Yaskawa INFORM job: KRIS1(-160_-90)07.JBI

/JOB
//NAME KRIS1(-160_-90)07
//POS
///NPOS 268,268,268,15,0,0
///TOOL 0
///POSTYPE PULSE
///PULSE
C00000=-1357,-104031,-113776,9484,62521,80538
C00001=-1357,-104031,-113776,9484,62521,80538
C00002=-36470,-76528,-106815,19279,71473,77234
C00003=-134470,-76528,-106815,19279,71473,77234
C00004=-174981,-50493,-90161,40064,84672,66854
C00005=-187879,-63712,-94262,49080,81916,61249
C00006=-186060,-71155,-91964,59790,82905,66762
C00007=-178869,-72848,-88692,57971,77164,66872
C00008=-178869,-73293,-87273,58169,76560,66435
C00009=-178869,-73560,-86246,58315,76140,66130
C00010=-178674,-73111,-86205,58218,76137,66246
C00011=-177360,-70267,-84836,57702,75706,66732
C00012=-178674,-73111,-86205,58218,76137,66246
C00013=-178674,-71838,-89995,57689,77779,67427
C00014=-187879,-63712,-94262,49080,81916,61249
C00015=-188382,-49930,-83952,49213,82654,61403
C00016=-188014,-50962,-81654,49243,81175,60803
C00017=-188014,-51673,-80691,49342,80537,60470
C00018=-188014,-51583,-80818,49329,80620,60513
C00019=-186548,-48975,-79328,48719,80176,60967
C00020=-188014,-51583,-80818,49329,80620,60513
C00021=-188014,-47372,-85350,48920,83933,62231
C00022=-182062,-62332,-92296,30199,64588,50507
C00023=-184090,-61700,-84500,30217,57788,46513
C00024=-184090,-62275,-83323,30540,56902,46238
C00025=-184090,-62207,-83473,30499,57013,46272
C00026=-182547,-59219,-81900,29317,56990,46927
C00027=-184090,-62207,-83473,30499,57013,46272
C00028=-182062,-62332,-92296,30199,64588,50507
C00029=-213458,-81436,-127572,45024,85737,46387
C00030=-213462,-137262,-127618,80891,60645,46377
C00031=-213462,-137262,-127618,80891,60645,46377
C00032=-213462,-137262,-127281,45256,60365,46369
C00033=-190178,-104312,-111371,30656,55898,55861
C00034=-182510,-123951,-113302,29184,45443,56133
C00035=-182510,-123446,-111392,29630,44641,55847
C00036=-182510,-123495,-111565,29589,44713,55873
C00037=-180510,-119420,-110276,27514,45182,57098
C00038=-182510,-123495,-111565,29589,44713,55873
C00039=-182510,-124409,-115363,28705,46354,56443
C00040=-219776,-105077,-106077,50090,64862,45838
C00041=-220601,-99189,-101769,50266,65553,45786
C00042=-220601,-99263,-100237,50600,64914,45410
C00043=-220601,-99258,-100424,50559,64990,45455
C00044=-218392,-97957,-99927,49618,64034,46123
C00045=-220601,-99258,-100424,50559,64990,45455
C00046=-219776,-105077,-106077,50090,64862,45838
C00047=-190178,-104312,-111371,30656,55898,55861
C00048=-229240,-109114,-135810,47014,82062,49329
C00049=-229240,-109114,-135810,47014,82062,49329
C00050=-195224,-66819,-119592,28790,78815,60275
C00051=-159578,-94739,-111578,14965,102577,71346
C00052=-157566,-87256,-71357,3912,80960,68626
C00053=-158237,-87274,-67249,3997,78461,68317
C00054=-158512,-86753,-64553,4040,77085,68177
C00055=-158512,-85902,-62577,4050,76306,68151
C00056=-159334,-88042,-63583,4126,75872,67853
C00057=-159947,-89575,-64280,4185,75546,67628
C00058=-158678,-86897,-63962,4060,76658,68106
C00059=-158401,-87046,-65688,4022,77628,68233
C00060=-157724,-87159,-69865,3934,80101,68545
C00061=-157573,-90681,-89077,3900,90084,68907
C00062=-157703,-92030,-92713,3898,91631,68910
C00063=-158377,-93978,-89476,3949,88678,68591
C00064=-158653,-94353,-86922,3974,86930,68442
C00065=-158653,-94065,-85585,3975,86257,68419
C00066=-158901,-94897,-86117,3998,86172,68332
C00067=-159738,-97484,-87119,4071,85502,68025
C00068=-158508,-94414,-86637,3961,86718,68485
C00069=-158233,-93872,-88035,3937,87841,68614
C00070=-157561,-92106,-91348,3883,90748,68930
C00071=-157550,-88189,-103730,3988,100358,69239
C00072=-157494,-88262,-105997,3987,101710,69297
C00073=-158163,-92718,-103752,3992,98079,68960
C00074=-158927,-96366,-102620,4029,95553,68625
C00075=-158927,-96520,-101690,4026,94903,68601
C00076=-158927,-96495,-101852,4026,95015,68605
C00077=-159979,-100458,-103367,4107,93966,68220
C00078=-158702,-95424,-101809,4010,95525,68699
C00079=-158425,-94019,-102865,4000,96880,68834
C00080=-157748,-89886,-105246,3989,100429,69172
C00081=-156260,-82084,-105550,20461,72444,69801
C00082=-137260,-84248,-120477,10166,77039,76482
C00083=-137260,-138866,-133764,10166,31487,76482
C00084=-31464,-162597,-133764,10166,12061,76482
C00085=11401,-148032,-125425,11667,35640,75771
C00086=126225,-114648,-117375,36487,17100,65054
C00087=160935,-140983,-109640,13468,75088,74332
C00088=169853,-118963,-84593,12681,69660,-86771
C00089=185015,-85467,-64977,10138,72568,-81037
C00090=186046,-86587,-63372,10054,70902,-80807
C00091=186046,-85672,-61299,10100,70108,-80875
C00092=186099,-85805,-61481,10085,70145,-80849
C00093=187639,-87511,-62050,9863,69435,-80354
C00094=183812,-88241,-67244,10331,72692,-81455
C00095=173907,-109296,-96285,11524,80966,-84205
C00096=165243,-81442,-84446,9619,88683,-83239
C00097=165243,-81286,-81084,9622,86723,-83389
C00098=165344,-81527,-80785,9608,86408,-83377
C00099=165344,-81401,-79599,9612,85752,-83428
C00100=165344,-81434,-79892,9611,85913,-83415
C00101=166373,-84175,-81092,9484,85132,-83124
C00102=163979,-82682,-81772,9785,86585,-83830
C00103=160654,-84295,-101618,10197,98198,-83833
C00104=158831,-94543,-102742,7696,93888,-81952
C00105=159073,-94488,-101668,7659,93239,-81911
C00106=159073,-94700,-100523,7653,92432,-81960
C00107=159073,-94669,-100714,7655,92565,-81952
C00108=160071,-98397,-102165,7522,91459,-81686
C00109=158831,-94357,-103427,7703,94400,-81921
C00110=161715,-86803,-103327,4886,98608,-77730
C00111=162141,-92472,-85533,-3463,86932,-68770
C00112=161818,-87798,-71417,-3733,80713,-68419
C00113=160875,-83714,-65601,-3665,79192,-68698
C00114=161375,-83882,-63363,-3725,77755,-68482
C00115=161375,-83186,-61665,-3733,77069,-68462
C00116=161375,-83302,-61946,-3731,77181,-68466
C00117=162606,-86103,-62964,-3849,76427,-68017
C00118=161375,-84160,-64056,-3722,78038,-68491
C00119=162005,-87841,-70029,-3758,79847,-68329
C00120=161949,-92223,-96357,-3744,93768,-68761
C00121=161804,-92637,-92737,-3704,91325,-68737
C00122=160782,-89227,-87327,-3611,89709,-69033
C00123=161425,-90912,-85851,-3665,87970,-68764
C00124=161425,-90690,-84578,-3665,87303,-68744
C00125=161425,-90728,-84781,-3665,87408,-68747
C00126=162412,-93603,-85938,-3751,86691,-68391
C00127=161425,-91016,-86520,-3665,88326,-68774
C00128=162058,-93372,-91608,-3722,90267,-68620
C00129=162002,-88104,-107646,-3859,102814,-69021
C00130=161873,-89540,-106233,-3806,101205,-69011
C00131=162580,-93883,-103932,-3818,97597,-68666
C00132=159915,-93477,-102438,-3577,96772,-69526
C00133=159915,-93839,-100899,-3567,95642,-69493
C00134=159915,-93799,-101099,-3568,95785,-69497
C00135=160794,-97042,-102371,-3639,94941,-69180
C00136=159915,-93165,-103472,-3585,97568,-69550
C00137=164885,-102201,-108421,-4002,96197,-67859
C00138=149595,-96211,-103761,-5489,101844,-74102
C00139=148895,-100989,-103442,-6283,96942,-74202
C00140=149006,-93113,-100988,-5479,101691,-74295
C00141=149599,-96300,-103483,-5484,101628,-74092
C00142=137295,-108190,-106060,-5698,94014,-77976
C00143=149608,-96287,-103789,-5489,101823,-74097
C00144=160720,-151449,-123129,-13814,72249,-68439
C00145=174899,-138237,-126795,1008,88740,-67536
C00146=163022,-96341,-102515,22398,105363,-76518
C00147=163017,-96713,-99258,22147,103326,-76913
C00148=166118,-105377,-102170,18852,96347,-77230
C00149=163022,-96736,-99152,22139,103253,-76925
C00150=162158,-93804,-96763,22109,103515,-77196
C00151=174925,-92085,-97088,18785,97864,-73864
C00152=167549,-101389,-103915,18999,98984,-76305
C00153=163194,-119427,-113025,19710,97619,-78016
C00154=163006,-95534,-87485,21597,97146,-78065
C00155=166449,-103981,-88986,17839,88165,-78380
C00156=167279,-118842,-91930,16839,77497,-71410
C00157=163006,-94576,-83573,21494,95359,-78388
C00158=162142,-91714,-81191,21448,95589,-78662
C00159=178049,-105864,-87645,15594,79224,-67328
C00160=171906,-113065,-93299,16245,80217,-69386
C00161=173072,-122981,-101575,-4997,88706,-65554
C00162=166636,-106884,-92426,-2568,94448,-67910
C00163=167630,-109607,-91139,-2502,92292,-67531
C00164=162194,-92631,-84353,657,102863,-69400
C00165=163060,-95514,-86735,782,102839,-69097
C00166=155875,-120106,-94474,-3152,88541,-71437
C00167=155875,-121766,-97691,-3153,89666,-71465
C00168=178442,-133591,-104623,-8068,82135,-63325
C00169=176542,-133362,-109369,-6755,86992,-64211
C00170=163036,-88875,-67291,2288,96831,-69180
C00171=159610,-85618,-62441,1680,95605,-70370
C00172=162086,-85813,-60042,2106,93969,-69554
C00173=162173,-84225,-60457,2128,95039,-69506
C00174=163038,-86971,-62872,2279,95091,-69211
C00175=151835,-92381,-62525,304,92274,-73022
C00176=151835,-95702,-69255,305,94709,-73016
C00177=163041,-94022,-81579,12660,98605,-75478
C00178=162985,-87715,-64806,21312,87868,-79725
C00179=162980,-85781,-60474,21324,86307,-80003
C00180=163244,-83528,-57038,21357,85347,-80079
C00181=162985,-85725,-60330,21325,86250,-80011
C00182=162122,-82990,-57905,21265,86391,-80297
C00183=171549,-75890,-53739,21771,84944,-77151
C00184=153122,-94015,-66237,20488,88162,-83220
C00185=168603,-127327,-105850,12339,78437,77405
C00186=149894,-144724,-110594,14594,75698,70467
C00187=126225,-114648,-117375,36487,17100,65054
C00188=118781,-153853,-134406,32592,23357,65054
C00189=12470,-167083,-125425,11667,16324,75771
C00190=-137258,-84249,-120477,10166,64820,76482
C00191=-160540,-100857,-113063,23155,68829,67581
C00192=-174981,-50493,-90161,40064,84672,66854
C00193=-187879,-63712,-94262,49080,81916,61249
C00194=-230671,-89591,-126680,64018,108053,56526
C00195=-230671,-150117,-126680,83924,107200,56526
C00196=-230671,-150117,-126680,83924,107200,56526
C00197=-230671,-150117,-126680,39809,88276,56526
C00198=-185677,-128245,-133585,38839,68006,71149
C00199=-143279,-154007,-127386,2438,36675,82296
C00200=-143590,-141394,-120265,2620,38778,82199
C00201=-143742,-142485,-120562,2786,38406,82105
C00202=-143590,-141570,-120589,2614,38886,82201
C00203=-202436,-119741,-113840,40114,62182,59763
C00204=-198557,-130318,-109753,40932,40025,50599
C00205=-196641,-131399,-103756,47310,28244,43457
C00206=-193242,-140218,-107458,47365,24899,43542
C00207=-143279,-154007,-127386,2438,36675,82296
C00208=-143372,-162538,-136969,2444,38193,82294
C00209=-143372,-162538,-136969,2444,38193,82294
C00210=-169193,-120980,-126540,32650,66176,77929
C00211=-162706,-113692,-115443,30259,61179,79142
C00212=-159565,-103232,-109234,28227,61475,80556
C00213=-143742,-142485,-120562,2786,38406,82105
C00214=-143590,-141570,-120589,2614,38886,82201
C00215=-133202,-124644,-116491,13354,48701,89198
C00216=-140045,-120904,-111840,33091,52219,88326
C00217=-147445,-115513,-104255,49921,56750,87686
C00218=-147948,-114087,-100063,56693,57074,88007
C00219=-151078,-112408,-101145,56872,59820,87990
C00220=-162706,-113692,-115443,30259,61179,79142
C00221=-169193,-120980,-126540,32650,66176,77929
C00222=-169193,-120980,-126540,32650,66176,77929
C00223=-169193,-120980,-126540,32650,66176,77929
C00224=-169193,-120980,-126540,32650,66176,77929
C00225=-189746,-144194,-133392,42604,68859,69788
C00226=-182215,-131283,-122466,40105,65254,71827
C00227=-178156,-121131,-115309,38344,64069,73249
C00228=-157379,-154126,-124637,33193,46204,76615
C00229=-155622,-153970,-121840,43876,49612,78686
C00230=-159534,-158630,-125101,47522,52653,77846
C00231=-179897,-166210,-133900,51769,64813,73191
C00232=-179897,-166210,-133900,51769,64813,73191
C00233=-179897,-166210,-133900,51769,64813,73191
C00234=-144017,-127352,-123370,33815,56946,88116
C00235=-136296,-120281,-120593,-4079,55650,85264
C00236=-135245,-107004,-113403,-4642,58094,85574
C00237=-145143,-100864,-111178,1649,59705,81829
C00238=-158741,-87238,-105999,9726,64424,77163
C00239=-147367,-98171,-102243,-17290,47874,78333
C00240=-144875,-102905,-108473,-14295,50590,79740
C00241=-136296,-120281,-120593,-4079,55650,85264
C00242=-138675,-113827,-131364,-2561,67962,83610
C00243=-184171,-107868,-119248,16468,98370,62097
C00244=-171634,-136713,-119987,14813,82155,64373
C00245=-158729,-95167,-103646,5818,103191,69841
C00246=-160167,-97375,-101626,5748,100928,69246
C00247=-158743,-95268,-103371,5812,102972,69826
C00248=-157888,-92366,-100981,5813,102933,70115
C00249=-149921,-107326,-105235,5663,97333,72568
C00250=-153886,-106740,-107354,5718,99208,71304
C00251=-163031,-143044,-118600,5591,88166,67691
C00252=-166711,-113552,-95038,4166,94777,66107
C00253=-164943,-103868,-87794,1353,97515,66988
C00254=-158755,-94787,-86481,-976,103949,69303
C00255=-157900,-91912,-84097,-841,103969,69603
C00256=-153517,-113616,-91125,2667,94271,70849
C00257=-153517,-115912,-96262,2679,96250,70891
C00258=-166250,-149525,-105399,1185,84912,66421
C00259=-160517,-92560,-68375,1999,97708,69937
C00260=-159946,-85824,-59096,2104,95443,70095
C00261=-158782,-86330,-62292,2348,97119,70521
C00262=-157926,-83586,-59872,2521,97014,70811
C00263=-149643,-92034,-61525,4148,93353,73521
C00264=-149643,-98229,-74267,4194,97999,73676
C00265=-159578,-94739,-111578,14965,102577,71346
C00266=-134470,-76528,-106815,19279,71473,77234
C00267=-36470,-76528,-106815,19279,71473,77234
BC00000=230677,678686,1075151
BC00001=230677,678686,1075151
BC00002=295325,674563,1075175
BC00003=353535,895977,1075175
BC00004=353024,938434,1075175
BC00005=352575,975666,1075175
BC00006=352579,975411,1075168
BC00007=352579,975411,1075168
BC00008=352579,975411,1075168
BC00009=352579,975411,1075168
BC00010=352579,975411,1075168
BC00011=352579,975411,1075168
BC00012=352579,975411,1075168
BC00013=352579,975411,1075168
BC00014=352575,975666,1075175
BC00015=352575,975666,1075175
BC00016=352575,975666,1075175
BC00017=352575,975666,1075175
BC00018=352575,975666,1075175
BC00019=352575,975666,1075172
BC00020=352575,975666,1075175
BC00021=352575,975666,1075175
BC00022=352575,975666,1075171
BC00023=352575,975666,1075171
BC00024=352575,975666,1075171
BC00025=352575,975666,1075171
BC00026=352575,975666,1075171
BC00027=352575,975666,1075171
BC00028=352575,975666,1075171
BC00029=352575,975666,1075171
BC00030=352575,975666,1075171
BC00031=265670,989358,1075171
BC00032=265670,989358,1075171
BC00033=265670,1007918,1075171
BC00034=265670,1007918,1075171
BC00035=265670,1007918,1075171
BC00036=265670,1007918,1075171
BC00037=265670,1007918,1075171
BC00038=265670,1007918,1075171
BC00039=265670,1007918,1075171
BC00040=265670,1036547,1075171
BC00041=265670,1036547,1075171
BC00042=265670,1036547,1075171
BC00043=265670,1036547,1075171
BC00044=265670,1036547,1075171
BC00045=265670,1036547,1075171
BC00046=265670,1036547,1075171
BC00047=265670,1007918,1075171
BC00048=288113,1006657,1075170
BC00049=288113,1006657,1075170
BC00050=366423,961968,1075170
BC00051=353535,975867,1075175
BC00052=382950,976989,1075175
BC00053=382950,976989,1075175
BC00054=382950,976989,1075175
BC00055=382950,976989,1075175
BC00056=382949,976988,1075174
BC00057=382949,976988,1075174
BC00058=382950,976989,1075175
BC00059=382950,976989,1075175
BC00060=382950,976989,1075175
BC00061=382631,988041,1075175
BC00062=382092,1006363,1075175
BC00063=382092,1006363,1075175
BC00064=382092,1006363,1075175
BC00065=382092,1006363,1075175
BC00066=382092,1006363,1075175
BC00067=382092,1006363,1075175
BC00068=382092,1006363,1075175
BC00069=382092,1006363,1075175
BC00070=382092,1006363,1075175
BC00071=382047,1017409,1075175
BC00072=382070,1033391,1075175
BC00073=382070,1033391,1075175
BC00074=382070,1033391,1075175
BC00075=382070,1033391,1075175
BC00076=382070,1033391,1075175
BC00077=382070,1033391,1075175
BC00078=382070,1033391,1075175
BC00079=382070,1033391,1075175
BC00080=382070,1033391,1075175
BC00081=381896,966588,1075175
BC00082=353816,923989,1075175
BC00083=353816,923989,1075175
BC00084=379773,1126391,1075175
BC00085=398190,1030285,1075175
BC00086=312632,1138057,1075175
BC00087=340753,1115300,1075175
BC00088=340766,1114848,1075175
BC00089=340766,1114848,1075175
BC00090=340766,1114848,1075175
BC00091=340766,1114848,1075175
BC00092=340766,1114848,1075175
BC00093=340766,1114848,1075175
BC00094=340766,1114848,1075175
BC00095=340766,1114848,1075175
BC00096=322874,1114287,1075175
BC00097=322874,1114287,1075175
BC00098=322874,1114287,1075175
BC00099=322874,1114287,1075175
BC00100=322874,1114287,1075175
BC00101=322874,1114287,1075175
BC00102=322874,1114287,1075175
BC00103=321868,1114200,1075175
BC00104=305323,1086030,1075175
BC00105=305323,1086030,1075175
BC00106=305323,1086030,1075175
BC00107=305323,1086030,1075175
BC00108=305323,1086030,1075175
BC00109=305323,1086030,1075175
BC00110=323405,1100688,1075175
BC00111=381464,1145987,1075175
BC00112=383295,1147007,1075175
BC00113=383295,1147007,1075175
BC00114=383295,1147007,1075175
BC00115=383295,1147007,1075175
BC00116=383295,1147007,1075175
BC00117=383295,1147007,1075175
BC00118=383295,1147007,1075175
BC00119=383295,1147007,1075175
BC00120=383362,1127243,1075175
BC00121=383252,1117196,1075175
BC00122=383252,1117196,1075175
BC00123=383252,1117196,1075175
BC00124=383252,1117196,1075175
BC00125=383252,1117196,1075175
BC00126=383252,1117196,1075175
BC00127=383252,1117196,1075175
BC00128=383252,1117196,1075175
BC00129=383208,1098974,1075175
BC00130=383049,1090382,1075175
BC00131=383049,1090382,1075175
BC00132=383049,1090382,1075175
BC00133=383049,1090382,1075175
BC00134=383049,1090382,1075175
BC00135=383049,1090382,1075175
BC00136=383049,1090382,1075175
BC00137=383049,1090382,1075175
BC00138=348637,1089204,1075175
BC00139=348912,1090234,1075175
BC00140=348912,1090234,1075175
BC00141=348912,1090234,1075175
BC00142=348912,1090234,1075175
BC00143=364565,1089242,1075175
BC00144=363879,1086668,1075175
BC00145=346096,1068466,1075175
BC00146=323525,1045363,1075175
BC00147=322819,1049711,1075175
BC00148=322608,1051010,1075175
BC00149=322536,1051450,1075175
BC00150=322536,1051450,1075175
BC00151=322608,1051010,1075175
BC00152=322608,1051010,1075175
BC00153=318232,1049352,1075175
BC00154=323451,1072164,1075175
BC00155=322745,1076512,1075175
BC00156=322745,1076512,1075175
BC00157=322462,1078251,1075175
BC00158=322462,1078251,1075175
BC00159=322745,1076512,1075175
BC00160=322745,1076512,1075175
BC00161=364639,1081055,1075175
BC00162=365322,1085072,1075175
BC00163=365322,1085072,1075175
BC00164=365595,1086678,1075175
BC00165=365595,1086678,1075175
BC00166=365322,1085072,1075175
BC00167=365322,1085072,1075175
BC00168=380567,1081094,1075175
BC00169=378567,1084057,1075175
BC00170=364571,1104797,1075175
BC00171=365253,1109149,1075175
BC00172=365253,1109149,1075175
BC00173=365525,1110890,1075175
BC00174=365525,1110890,1075175
BC00175=365253,1109149,1075175
BC00176=365253,1109149,1075175
BC00177=341083,1103324,1075175
BC00178=323368,1101944,1075175
BC00179=322661,1106292,1075175
BC00180=322661,1106292,1075175
BC00181=322379,1108032,1075175
BC00182=322379,1108032,1075175
BC00183=322661,1106292,1075175
BC00184=306985,1106255,1075175
BC00185=340753,1115300,1075175
BC00186=340753,1115300,1075175
BC00187=312632,1138057,1075175
BC00188=312632,1138057,1075175
BC00189=398190,1030285,1075175
BC00190=353817,923990,1075175
BC00191=381896,966588,1075175
BC00192=353024,938434,1075175
BC00193=352575,975666,1075175
BC00194=352575,975666,1075175
BC00195=269490,975666,1075175
BC00196=209516,997345,1075175
BC00197=229953,997345,1075175
BC00198=209516,997345,1075175
BC00199=209516,997345,1075175
BC00200=209516,997345,1075171
BC00201=209516,997345,1075171
BC00202=209516,997345,1075171
BC00203=234573,1028656,1075168
BC00204=234573,1028656,1075168
BC00205=234573,1028656,1075168
BC00206=234573,1028656,1075168
BC00207=209516,997345,1075175
BC00208=209517,887810,1075171
BC00209=304062,887810,1075171
BC00210=304062,986914,1075171
BC00211=304062,986914,1075171
BC00212=304062,986914,1075171
BC00213=209516,997345,1075171
BC00214=209516,997345,1075171
BC00215=304062,986914,1075171
BC00216=304062,986914,1075171
BC00217=304062,986914,1075171
BC00218=304062,986914,1075171
BC00219=304062,986914,1075171
BC00220=304062,986914,1075171
BC00221=304062,986914,1075171
BC00222=304062,879334,1075171
BC00223=206079,877704,1075171
BC00224=206079,986425,1075171
BC00225=216915,1007447,1075171
BC00226=216915,1007447,1075171
BC00227=216915,1007447,1075171
BC00228=216915,1007447,1075171
BC00229=216914,1007446,1075170
BC00230=216915,1007447,1075171
BC00231=216914,1007447,1075168
BC00232=216914,908506,1075168
BC00233=299617,908506,1075168
BC00234=274777,953856,1075168
BC00235=304062,986914,1075171
BC00236=304062,986914,1075171
BC00237=304062,986914,1075171
BC00238=304061,986914,1075167
BC00239=304062,986914,1075171
BC00240=304062,986914,1075171
BC00241=304062,986914,1075171
BC00242=308072,990794,1075171
BC00243=363636,1044565,1075175
BC00244=363636,1044565,1075175
BC00245=364364,1042023,1075175
BC00246=364654,1041006,1075172
BC00247=364655,1041006,1075175
BC00248=364655,1041006,1075175
BC00249=364654,1041006,1075172
BC00250=370115,1041376,1075173
BC00251=370115,1041376,1075173
BC00252=364161,1042499,1075173
BC00253=364434,1040968,1075174
BC00254=364774,1039056,1075175
BC00255=364774,1039056,1075175
BC00256=364434,1040968,1075174
BC00257=364434,1040968,1075174
BC00258=364434,1040968,1075174
BC00259=353535,1018425,1075175
BC00260=355520,1012445,1075175
BC00261=355520,1012445,1075175
BC00262=355520,1012445,1075175
BC00263=355520,1012445,1075175
BC00264=355520,1012445,1075175
BC00265=353535,975867,1075175
BC00266=353535,895977,1075175
BC00267=295325,674563,1075175
EC00000=12352,-24024
EC00001=-1418783,924
EC00002=-1418945,-556475
EC00003=-1418945,-556475
EC00004=-1342906,-556475
EC00005=-1276223,-556475
EC00006=-1276676,-556475
EC00007=-1276676,-556475
EC00008=-1276676,-556475
EC00009=-1276676,-556475
EC00010=-1276676,-556475
EC00011=-1276676,-556475
EC00012=-1276676,-556475
EC00013=-1276676,-556475
EC00014=-1276223,-556475
EC00015=-1276223,-556475
EC00016=-1276223,-556475
EC00017=-1276223,-556475
EC00018=-1276223,-556475
EC00019=-1276222,-556475
EC00020=-1276223,-556475
EC00021=-1276223,-556475
EC00022=-1276222,-556476
EC00023=-1276222,-556476
EC00024=-1276222,-556476
EC00025=-1276222,-556476
EC00026=-1276222,-556476
EC00027=-1276222,-556476
EC00028=-1276222,-556476
EC00029=-1276222,-556476
EC00030=-1276222,-556476
EC00031=-1276222,-556476
EC00032=-1276222,-556476
EC00033=-1276222,-556476
EC00034=-1276222,-556476
EC00035=-1276222,-556476
EC00036=-1276222,-556476
EC00037=-1276222,-556476
EC00038=-1276222,-556476
EC00039=-1276222,-556476
EC00040=-1276222,-556476
EC00041=-1276222,-556476
EC00042=-1276222,-556476
EC00043=-1276222,-556476
EC00044=-1276222,-556476
EC00045=-1276222,-556476
EC00046=-1276222,-556476
EC00047=-1276222,-556476
EC00048=-1276222,-556476
EC00049=-1276222,-556476
EC00050=-1276222,-556476
EC00051=-1418945,-556475
EC00052=-1418945,-556475
EC00053=-1418945,-556475
EC00054=-1418945,-556475
EC00055=-1418945,-556475
EC00056=-1418943,-556475
EC00057=-1418943,-556475
EC00058=-1418945,-556475
EC00059=-1418945,-556475
EC00060=-1418945,-556475
EC00061=-1418945,-556475
EC00062=-1418945,-556475
EC00063=-1418945,-556475
EC00064=-1418945,-556475
EC00065=-1418945,-556475
EC00066=-1418945,-556475
EC00067=-1418945,-556475
EC00068=-1418945,-556475
EC00069=-1418945,-556475
EC00070=-1418945,-556475
EC00071=-1418945,-556475
EC00072=-1418945,-556475
EC00073=-1418945,-556475
EC00074=-1418945,-556475
EC00075=-1418945,-556475
EC00076=-1418945,-556475
EC00077=-1418945,-556475
EC00078=-1418945,-556475
EC00079=-1418945,-556475
EC00080=-1418945,-556475
EC00081=-1418945,-556475
EC00082=-1418945,-556475
EC00083=-1418945,-556475
EC00084=-1418945,-556475
EC00085=-1595090,-3837
EC00086=-1773681,556475
EC00087=-1773681,556475
EC00088=-1773681,556475
EC00089=-1773681,556475
EC00090=-1773681,556475
EC00091=-1773681,556475
EC00092=-1773681,556475
EC00093=-1773681,556475
EC00094=-1773681,556475
EC00095=-1773681,556475
EC00096=-1773681,556475
EC00097=-1773681,556475
EC00098=-1773681,556475
EC00099=-1773681,556475
EC00100=-1773681,556475
EC00101=-1773681,556475
EC00102=-1773681,556475
EC00103=-1773681,556475
EC00104=-1773681,556475
EC00105=-1773681,556475
EC00106=-1773681,556475
EC00107=-1773681,556475
EC00108=-1773681,556475
EC00109=-1773681,556475
EC00110=-1773681,556475
EC00111=-1773681,556475
EC00112=-1773681,556475
EC00113=-1773681,556475
EC00114=-1773681,556475
EC00115=-1773681,556475
EC00116=-1773681,556475
EC00117=-1773681,556475
EC00118=-1773681,556475
EC00119=-1773681,556475
EC00120=-1773681,556475
EC00121=-1773681,556475
EC00122=-1773681,556475
EC00123=-1773681,556475
EC00124=-1773681,556475
EC00125=-1773681,556475
EC00126=-1773681,556475
EC00127=-1773681,556475
EC00128=-1773681,556475
EC00129=-1773681,556475
EC00130=-1773681,556475
EC00131=-1773681,556475
EC00132=-1773681,556475
EC00133=-1773681,556475
EC00134=-1773681,556475
EC00135=-1773681,556475
EC00136=-1773681,556475
EC00137=-1773681,556475
EC00138=-1773681,556475
EC00139=-1773681,556475
EC00140=-1773681,556475
EC00141=-1773681,556475
EC00142=-1773681,556475
EC00143=-1773681,556475
EC00144=-1773681,556475
EC00145=-1773681,556475
EC00146=-1773681,556475
EC00147=-1773681,556475
EC00148=-1773681,556475
EC00149=-1773681,556475
EC00150=-1773681,556475
EC00151=-1773681,556475
EC00152=-1773681,556475
EC00153=-1773681,556475
EC00154=-1773681,556475
EC00155=-1773681,556475
EC00156=-1773681,556475
EC00157=-1773681,556475
EC00158=-1773681,556475
EC00159=-1773681,556475
EC00160=-1773681,556475
EC00161=-1773681,556475
EC00162=-1773681,556475
EC00163=-1773681,556475
EC00164=-1773681,556475
EC00165=-1773681,556475
EC00166=-1773681,556475
EC00167=-1773681,556475
EC00168=-1773681,556475
EC00169=-1773681,556475
EC00170=-1773681,556475
EC00171=-1773681,556475
EC00172=-1773681,556475
EC00173=-1773681,556475
EC00174=-1773681,556475
EC00175=-1773681,556475
EC00176=-1773681,556475
EC00177=-1773681,556475
EC00178=-1773681,556475
EC00179=-1773681,556475
EC00180=-1773681,556475
EC00181=-1773681,556475
EC00182=-1773681,556475
EC00183=-1773681,556475
EC00184=-1773681,556475
EC00185=-1773681,556475
EC00186=-1773681,556475
EC00187=-1773681,556475
EC00188=-1773681,556475
EC00189=-1595090,-3837
EC00190=-1418947,-556468
EC00191=-1418945,-556475
EC00192=-1342906,-556475
EC00193=-1276223,-556475
EC00194=-1276223,-556475
EC00195=-1276223,-556475
EC00196=-1276223,-556475
EC00197=-1276223,-556475
EC00198=-1276223,-556475
EC00199=-1276223,-556475
EC00200=-1276222,-556475
EC00201=-1276222,-556475
EC00202=-1276222,-556475
EC00203=-1276221,-556475
EC00204=-1276221,-556475
EC00205=-1276221,-556475
EC00206=-1276221,-556475
EC00207=-1276223,-556475
EC00208=-1276222,-556475
EC00209=-1276222,-556475
EC00210=-1276222,-556475
EC00211=-1276222,-556475
EC00212=-1276222,-556475
EC00213=-1276222,-556475
EC00214=-1276222,-556475
EC00215=-1276222,-556475
EC00216=-1276222,-556475
EC00217=-1276222,-556475
EC00218=-1276222,-556475
EC00219=-1276222,-556475
EC00220=-1276222,-556475
EC00221=-1276222,-556475
EC00222=-1276222,-556475
EC00223=-1276222,-556475
EC00224=-1276222,-556475
EC00225=-1276222,-556475
EC00226=-1276222,-556475
EC00227=-1276222,-556475
EC00228=-1276222,-556475
EC00229=-1276221,-556476
EC00230=-1276222,-556475
EC00231=-1276221,-556475
EC00232=-1276221,-556475
EC00233=-1276221,-556475
EC00234=-1276221,-556475
EC00235=-1276222,-556475
EC00236=-1276222,-556475
EC00237=-1276222,-556475
EC00238=-1276222,-556476
EC00239=-1276222,-556475
EC00240=-1276222,-556475
EC00241=-1276222,-556475
EC00242=-1285829,-556475
EC00243=-1418945,-556475
EC00244=-1418945,-556475
EC00245=-1418945,-556475
EC00246=-1418945,-556475
EC00247=-1418945,-556475
EC00248=-1418945,-556475
EC00249=-1418945,-556475
EC00250=-1418945,-556475
EC00251=-1418945,-556475
EC00252=-1418944,-556475
EC00253=-1418944,-556475
EC00254=-1418945,-556475
EC00255=-1418945,-556475
EC00256=-1418944,-556475
EC00257=-1418944,-556475
EC00258=-1418944,-556475
EC00259=-1418945,-556475
EC00260=-1418945,-556475
EC00261=-1418945,-556475
EC00262=-1418945,-556475
EC00263=-1418945,-556475
EC00264=-1418945,-556475
EC00265=-1418945,-556475
EC00266=-1418945,-556475
EC00267=-1418945,-556475
///POSTYPE BASE
///RECTAN
///RCONF 0,0,0,0,0,0,0,0,0,0,0,0,0,0,0,0,0,0,0,0,0,0,0,0
P00006=0.222,-3.123,-1.508,0.0000,0.0000,0.0000
P00021=-0.225,-6.128,-0.405,0.0000,0.0000,0.0000
P00022=0.222,-3.123,-1.508,0.0000,0.0000,0.0000
P00023=0.143,-0.036,0.682,0.0000,0.0000,0.0000
P00031=1.853,-0.001,-1.549,0.0000,0.0000,0.0000
P00032=1.957,0.503,-7.217,0.0000,0.0000,0.0000
///RCONF 0,0,0,0,1,0,0,0,0,0,0,0,0,0,0,0,0,0,0,0,0,0,0,0
P00033=-0.123,0.612,-5.012,0.0000,0.0000,0.0000
///RCONF 0,0,0,0,0,0,0,0,0,0,0,0,0,0,0,0,0,0,0,0,0,0,0,0
P00034=-0.304,0.773,-2.693,0.0000,0.0000,0.0000
P00035=2.817,0.591,-1.622,0.0000,0.0000,0.0000
P00036=-1.108,-0.829,1.850,0.0000,0.0000,0.0000
P00051=0.367,3.892,0.009,0.0000,0.0000,0.0000
P00052=0.088,2.832,-0.342,0.0000,0.0000,0.0000
P00053=0.134,6.594,0.107,0.0000,0.0000,0.0000
P00054=-0.103,6.509,-0.702,0.0000,0.0000,0.0000
P00055=-0.342,8.912,1.324,0.0000,0.0000,0.0000
//INST
///DATE 2024/05/16 21:58
///ATTR SC,RW
///GROUP1 RB1,BS1
///GROUP2 ST1
NOP
SFTOF
SSFTOF
SFTOF3D
'OK_r2_O7.1(P)(-160.-90)
MOVJ C00000 BC00000 VJ=100.00  +MOVJ EC00000 VJ=100.00
MOVJ C00001 BC00001 VJ=100.00  +MOVJ EC00001 VJ=100.00
MOVJ C00002 BC00002 VJ=100.00  +MOVJ EC00002 VJ=100.00
MOVJ C00003 BC00003 VJ=100.00  +MOVJ EC00003 VJ=100.00
MOVJ C00004 BC00004 VJ=50.00  +MOVJ EC00004 VJ=50.00
MOVJ C00005 BC00005 VJ=50.00  +MOVJ EC00005 VJ=50.00
'DODAC SEARCH NO NOWA SPOINE
MOVL C00006 BC00006 V=400.0  +MOVJ EC00006 VJ=100.00
SMOVL C00007 BC00007 V=400.0  +MOVJ EC00007
SFTOF3D
SMOVL C00008 BC00008 V=100.0  +MOVJ EC00008
SREFP 3 C00009 BC00009  +REFP EC00009
CALL JOB:SEARCH-R1-S13D
SET P051 P006
SFTON3D P051
SMOVL C00010 BC00010 V=100.0  +MOVJ EC00010
SREFP 3 C00011 BC00011  +REFP EC00011
CALL JOB:SEARCH-R1-S13D
SET P051 P006
SFTON3D P051
SMOVL C00012 BC00012 V=100.0  +MOVJ EC00012
MOVL C00013 BC00013 V=400.0  +MOVJ EC00013 VJ=100.00
MOVL C00014 BC00014 V=400.0  +MOVJ EC00014 VJ=100.00
SFTOF3D
MOVL C00015 BC00015 V=400.0  +MOVJ EC00015 VJ=100.00
SMOVL C00016 BC00016 V=100.0  +MOVJ EC00016
SREFP 3 C00017 BC00017  +REFP EC00017
CALL JOB:SEARCH-R1-S13D
SET P052 P006
SFTON3D P052
SMOVL C00018 BC00018 V=100.0  +MOVJ EC00018
SREFP 3 C00019 BC00019  +REFP EC00019
CALL JOB:SEARCH-R1-S13D
SET P052 P006
SFTON3D P052
SMOVL C00020 BC00020 V=100.0  +MOVJ EC00020
MOVL C00021 BC00021 V=400.0  +MOVJ EC00021 VJ=100.00
SFTOF3D
MOVL C00022 BC00022 V=400.0  +MOVJ EC00022 VJ=100.00
SMOVL C00023 BC00023 V=100.0  +MOVJ EC00023
SREFP 3 C00024 BC00024  +REFP EC00024
CALL JOB:SEARCH-R1-S13D
SET P053 P006
SFTON3D P053
SMOVL C00025 BC00025 V=100.0  +MOVJ EC00025
SREFP 3 C00026 BC00026  +REFP EC00026
CALL JOB:SEARCH-R1-S13D
SET P053 P006
SFTON3D P053
SMOVL C00027 BC00027 V=100.0  +MOVJ EC00027
MOVL C00028 BC00028 V=400.0  +MOVJ EC00028 VJ=100.00
SFTOF3D
MOVL C00029 BC00029 V=400.0  +MOVJ EC00029 VJ=100.00
MOVL C00030 BC00030 V=400.0  +MOVJ EC00030 VJ=100.00
MOVL C00031 BC00031 V=400.0  +MOVJ EC00031 VJ=100.00
MOVL C00032 BC00032 V=400.0  +MOVJ EC00032 VJ=100.00
SFTOF3D
MOVL C00033 BC00033 V=400.0  +MOVJ EC00033 VJ=100.00
SMOVL C00034 BC00034 V=100.0  +MOVJ EC00034
SREFP 3 C00035 BC00035  +REFP EC00035
CALL JOB:SEARCH-R1-S13D
SET P054 P006
SFTON3D P054
SMOVL C00036 BC00036 V=100.0  +MOVJ EC00036
SREFP 3 C00037 BC00037  +REFP EC00037
CALL JOB:SEARCH-R1-S13D
SET P054 P006
SFTON3D P054
SMOVL C00038 BC00038 V=100.0  +MOVJ EC00038
MOVL C00039 BC00039 V=400.0  +MOVJ EC00039 VJ=100.00
SFTOF3D
MOVL C00040 BC00040 V=400.0  +MOVJ EC00040 VJ=100.00
SMOVL C00041 BC00041 V=100.0  +MOVJ EC00041
SREFP 3 C00042 BC00042  +REFP EC00042
CALL JOB:SEARCH-R1-S13D
SET P055 P006
SFTON3D P055
SMOVL C00043 BC00043 V=100.0  +MOVJ EC00043
SREFP 3 C00044 BC00044  +REFP EC00044
CALL JOB:SEARCH-R1-S13D
SET P055 P006
SFTON3D P055
SMOVL C00045 BC00045 V=100.0  +MOVJ EC00045
MOVL C00046 BC00046 V=400.0  +MOVJ EC00046 VJ=100.00
SFTOF3D
MOVL C00047 BC00047 V=400.0  +MOVJ EC00047 VJ=100.00
MOVL C00048 BC00048 V=400.0  +MOVJ EC00048 VJ=100.00
MOVL C00049 BC00049 V=400.0  +MOVJ EC00049 VJ=100.00
MOVL C00050 BC00050 V=400.0  +MOVJ EC00050 VJ=100.00
MOVJ C00051 BC00051 VJ=100.00  +MOVJ EC00051 VJ=100.00
'Path S1422
SFTOF3D
MOVJ C00052 BC00052 VJ=100.00  +MOVJ EC00052 VJ=100.00
MOVL C00053 BC00053 V=400.0  +MOVJ EC00053 VJ=100.00
SMOVL C00054 BC00054 V=100.0  +MOVJ EC00054
SREFP 3 C00055 BC00055  +REFP EC00055
CALL JOB:SEARCH-R1-S13D
SET P021 P006
SFTON3D P021
SMOVL C00056 BC00056 V=100.0  +MOVJ EC00056
SREFP 3 C00057 BC00057  +REFP EC00057
CALL JOB:SEARCH-R1-S13D
SET P021 P006
SFTON3D P021
SMOVL C00058 BC00058 V=100.0  +MOVJ EC00058
MOVL C00059 BC00059 V=400.0  +MOVJ EC00059 VJ=100.00
MOVL C00060 BC00060 V=1000.0  +MOVJ EC00060 VJ=100.00
MOVJ C00061 BC00061 VJ=100.00  +MOVJ EC00061 VJ=100.00
'Path S1423
SFTOF3D
MOVJ C00062 BC00062 VJ=100.00  +MOVJ EC00062 VJ=100.00
MOVL C00063 BC00063 V=400.0  +MOVJ EC00063 VJ=100.00
SMOVL C00064 BC00064 V=100.0  +MOVJ EC00064
SREFP 3 C00065 BC00065  +REFP EC00065
CALL JOB:SEARCH-R1-S13D
SET P022 P006
SFTON3D P022
SMOVL C00066 BC00066 V=100.0  +MOVJ EC00066
SREFP 3 C00067 BC00067  +REFP EC00067
CALL JOB:SEARCH-R1-S13D
SET P022 P006
SFTON3D P022
SMOVL C00068 BC00068 V=100.0  +MOVJ EC00068
MOVL C00069 BC00069 V=400.0  +MOVJ EC00069 VJ=100.00
MOVL C00070 BC00070 V=1000.0  +MOVJ EC00070 VJ=100.00
MOVJ C00071 BC00071 VJ=100.00  +MOVJ EC00071 VJ=100.00
'Path S1424
SFTOF3D
MOVJ C00072 BC00072 VJ=100.00  +MOVJ EC00072 VJ=100.00
MOVL C00073 BC00073 V=400.0  +MOVJ EC00073 VJ=100.00
SMOVL C00074 BC00074 V=100.0  +MOVJ EC00074
SREFP 3 C00075 BC00075  +REFP EC00075
CALL JOB:SEARCH-R1-S13D
SET P023 P006
SFTON3D P023
SMOVL C00076 BC00076 V=100.0  +MOVJ EC00076
SREFP 3 C00077 BC00077  +REFP EC00077
CALL JOB:SEARCH-R1-S13D
SET P023 P006
SFTON3D P023
SMOVL C00078 BC00078 V=100.0  +MOVJ EC00078
MOVL C00079 BC00079 V=400.0  +MOVJ EC00079 VJ=100.00
MOVL C00080 BC00080 V=1000.0  +MOVJ EC00080 VJ=100.00
'obrot
MOVJ C00081 BC00081 VJ=100.00  +MOVJ EC00081 VJ=100.00
MOVJ C00082 BC00082 VJ=100.00  +MOVJ EC00082 VJ=100.00
MOVJ C00083 BC00083 VJ=100.00  +MOVJ EC00083 VJ=100.00
MOVJ C00084 BC00084 VJ=100.00  +MOVJ EC00084 VJ=100.00
MOVJ C00085 BC00085 VJ=100.00  +MOVJ EC00085 VJ=100.00
MOVJ C00086 BC00086 VJ=100.00  +MOVJ EC00086 VJ=100.00
MOVJ C00087 BC00087 VJ=100.00  +MOVJ EC00087 VJ=100.00
'Path S1077
SFTOF3D
MOVJ C00088 BC00088 VJ=100.00  +MOVJ EC00088 VJ=100.00
MOVL C00089 BC00089 V=400.0  +MOVJ EC00089 VJ=100.00
SMOVL C00090 BC00090 V=100.0  +MOVJ EC00090
SREFP 3 C00091 BC00091  +REFP EC00091
CALL JOB:SEARCH-R1-S13D
SET P031 P006
SFTON3D P031
SMOVL C00092 BC00092 V=100.0  +MOVJ EC00092
SREFP 3 C00093 BC00093  +REFP EC00093
CALL JOB:SEARCH-R1-S13D
SET P031 P006
SFTON3D P031
SMOVL C00094 BC00094 V=100.0  +MOVJ EC00094
MOVL C00095 BC00095 V=1000.0  +MOVJ EC00095 VJ=100.00
MOVJ C00096 BC00096 VJ=100.00  +MOVJ EC00096 VJ=100.00
'Path S1078
SFTOF3D
MOVL C00097 BC00097 V=400.0  +MOVJ EC00097 VJ=100.00
SMOVL C00098 BC00098 V=100.0  +MOVJ EC00098
SREFP 3 C00099 BC00099  +REFP EC00099
CALL JOB:SEARCH-R1-S13D
SET P032 P006
SFTON3D P032
SMOVL C00100 BC00100 V=100.0  +MOVJ EC00100
SREFP 3 C00101 BC00101  +REFP EC00101
CALL JOB:SEARCH-R1-S13D
SET P032 P006
SFTON3D P032
SMOVL C00102 BC00102 V=100.0  +MOVJ EC00102
MOVL C00103 BC00103 V=1000.0  +MOVJ EC00103 VJ=100.00
'Path S1079
SFTOF3D
MOVL C00104 BC00104 V=400.0  +MOVJ EC00104 VJ=100.00
SMOVL C00105 BC00105 V=100.0  +MOVJ EC00105
SREFP 3 C00106 BC00106  +REFP EC00106
CALL JOB:SEARCH-R1-S13D
SET P033 P006
SFTON3D P033
SMOVL C00107 BC00107 V=100.0  +MOVJ EC00107
SREFP 3 C00108 BC00108  +REFP EC00108
CALL JOB:SEARCH-R1-S13D
SET P033 P006
SFTON3D P033
SMOVL C00109 BC00109 V=100.0  +MOVJ EC00109
MOVJ C00110 BC00110 VJ=100.00  +MOVJ EC00110 VJ=100.00
MOVJ C00111 BC00111 VJ=100.00  +MOVJ EC00111 VJ=100.00
'Path S1080
SFTOF3D
MOVJ C00112 BC00112 VJ=100.00  +MOVJ EC00112 VJ=100.00
MOVL C00113 BC00113 V=400.0  +MOVJ EC00113 VJ=100.00
SMOVL C00114 BC00114 V=100.0  +MOVJ EC00114
SREFP 3 C00115 BC00115  +REFP EC00115
CALL JOB:SEARCH-R1-S13D
SET P034 P006
SFTON3D P034
SMOVL C00116 BC00116 V=100.0  +MOVJ EC00116
SREFP 3 C00117 BC00117  +REFP EC00117
CALL JOB:SEARCH-R1-S13D
SET P034 P006
SFTON3D P034
SMOVL C00118 BC00118 V=100.0  +MOVJ EC00118
MOVL C00119 BC00119 V=1000.0  +MOVJ EC00119 VJ=100.00
MOVJ C00120 BC00120 VJ=100.00  +MOVJ EC00120 VJ=100.00
'Path S1081
SFTOF3D
MOVJ C00121 BC00121 VJ=100.00  +MOVJ EC00121 VJ=100.00
MOVL C00122 BC00122 V=400.0  +MOVJ EC00122 VJ=100.00
SMOVL C00123 BC00123 V=100.0  +MOVJ EC00123
SREFP 3 C00124 BC00124  +REFP EC00124
CALL JOB:SEARCH-R1-S13D
SET P035 P006
SFTON3D P035
SMOVL C00125 BC00125 V=100.0  +MOVJ EC00125
SREFP 3 C00126 BC00126  +REFP EC00126
CALL JOB:SEARCH-R1-S13D
SET P035 P006
SFTON3D P035
SMOVL C00127 BC00127 V=100.0  +MOVJ EC00127
MOVL C00128 BC00128 V=1000.0  +MOVJ EC00128 VJ=100.00
MOVJ C00129 BC00129 VJ=100.00  +MOVJ EC00129 VJ=100.00
'Path S1082
SFTOF3D
MOVJ C00130 BC00130 VJ=100.00  +MOVJ EC00130 VJ=100.00
MOVL C00131 BC00131 V=400.0  +MOVJ EC00131 VJ=100.00
SMOVL C00132 BC00132 V=100.0  +MOVJ EC00132
SREFP 3 C00133 BC00133  +REFP EC00133
CALL JOB:SEARCH-R1-S13D
SET P036 P006
SFTON3D P036
SMOVL C00134 BC00134 V=100.0  +MOVJ EC00134
SREFP 3 C00135 BC00135  +REFP EC00135
CALL JOB:SEARCH-R1-S13D
SET P036 P006
SFTON3D P036
SMOVL C00136 BC00136 V=133.3  +MOVJ EC00136
MOVL C00137 BC00137 V=400.0  +MOVJ EC00137 VJ=100.00
'Path W260
SFTOF3D
SFTON3D P036
SMOVL C00138 BC00138 V=400.0  +MOVJ EC00138
SMOVL C00139 BC00139 V=166.7 PL=0  +MOVJ EC00139
SREFP 1 C00140 BC00140  +REFP EC00140
SREFP 2 C00141 BC00141  +REFP EC00141
MACRO1 MJ#(0) ARGF14
ARCON
SMOVL C00142 BC00142 V=10.0  +MOVJ EC00142
ARCOF
SMOVL C00143 BC00143 V=400.0  +MOVJ EC00143
SMOVL C00144 BC00144 V=1000.0  +MOVJ EC00144
SFTOF3D
MOVJ C00145 BC00145 VJ=100.00  +MOVJ EC00145 VJ=100.00
'Path W261
SFTOF3D
SFTON3D P033
MOVJ C00146 BC00146 VJ=100.00  +MOVJ EC00146 VJ=100.00
SMOVL C00147 BC00147 V=400.0  +MOVJ EC00147
SMOVL C00148 BC00148 V=133.3 PL=0  +MOVJ EC00148
SREFP 1 C00149 BC00149  +REFP EC00149
SREFP 2 C00150 BC00150  +REFP EC00150
MACRO1 MJ#(0) ARGF14
ARCON
SMOVL C00151 BC00151 V=10.0  +MOVJ EC00151
ARCOF
SMOVL C00152 BC00152 V=400.0  +MOVJ EC00152
SMOVL C00153 BC00153 V=1000.0  +MOVJ EC00153
SFTOF3D
'Path W1083
SFTOF3D
SFTON3D P032
MOVJ C00154 BC00154 VJ=100.00  +MOVJ EC00154 VJ=100.00
SMOVL C00155 BC00155 V=400.0  +MOVJ EC00155
SMOVL C00156 BC00156 V=133.3 PL=0  +MOVJ EC00156
SREFP 1 C00157 BC00157  +REFP EC00157
SREFP 2 C00158 BC00158  +REFP EC00158
MACRO1 MJ#(0) ARGF14
ARCON
SMOVL C00159 BC00159 V=10.0  +MOVJ EC00159
ARCOF
SMOVL C00160 BC00160 V=400.0  +MOVJ EC00160
SFTOF3D
'Path W262
SFTOF3D
SFTON3D P035
MOVJ C00161 BC00161 VJ=100.00  +MOVJ EC00161 VJ=100.00
SMOVL C00162 BC00162 V=400.0  +MOVJ EC00162
SMOVL C00163 BC00163 V=133.3 PL=0  +MOVJ EC00163
SREFP 1 C00164 BC00164  +REFP EC00164
SREFP 2 C00165 BC00165  +REFP EC00165
MACRO1 MJ#(0) ARGF14
ARCON
SMOVL C00166 BC00166 V=10.0  +MOVJ EC00166
ARCOF
SMOVL C00167 BC00167 V=400.0  +MOVJ EC00167
SMOVL C00168 BC00168 V=1000.0  +MOVJ EC00168
SFTOF3D
MOVJ C00169 BC00169 VJ=100.00  +MOVJ EC00169 VJ=100.00
'Path W264
SFTOF3D
SFTON3D P034
MOVJ C00170 BC00170 VJ=100.00  +MOVJ EC00170 VJ=100.00
SMOVL C00171 BC00171 V=400.0  +MOVJ EC00171
SMOVL C00172 BC00172 V=100.0 PL=0  +MOVJ EC00172
SREFP 1 C00173 BC00173  +REFP EC00173
SREFP 2 C00174 BC00174  +REFP EC00174
MACRO1 MJ#(0) ARGF14
ARCON
SMOVL C00175 BC00175 V=10.0  +MOVJ EC00175
ARCOF
SMOVL C00176 BC00176 V=400.0  +MOVJ EC00176
SFTOF3D
MOVJ C00177 BC00177 VJ=100.00  +MOVJ EC00177 VJ=100.00
'Path W263
SFTOF3D
SFTON3D P031
MOVJ C00178 BC00178 VJ=100.00  +MOVJ EC00178 VJ=100.00
SMOVL C00179 BC00179 V=400.0  +MOVJ EC00179
SMOVL C00180 BC00180 V=133.3 PL=0  +MOVJ EC00180
SREFP 1 C00181 BC00181  +REFP EC00181
SREFP 2 C00182 BC00182  +REFP EC00182
MACRO1 MJ#(0) ARGF14
ARCON
SMOVL C00183 BC00183 V=10.0  +MOVJ EC00183
ARCOF
SMOVL C00184 BC00184 V=400.0  +MOVJ EC00184
SFTOF3D
'obrot
MOVJ C00185 BC00185 VJ=100.00  +MOVJ EC00185 VJ=100.00
MOVJ C00186 BC00186 VJ=100.00  +MOVJ EC00186 VJ=100.00
MOVJ C00187 BC00187 VJ=100.00  +MOVJ EC00187 VJ=100.00
MOVJ C00188 BC00188 VJ=100.00  +MOVJ EC00188 VJ=100.00
MOVJ C00189 BC00189 VJ=100.00  +MOVJ EC00189 VJ=100.00
MOVJ C00190 BC00190 VJ=100.00  +MOVJ EC00190 VJ=100.00
MOVJ C00191 BC00191 VJ=100.00  +MOVJ EC00191 VJ=100.00
MOVJ C00192 BC00192 VJ=50.00  +MOVJ EC00192 VJ=50.00
MOVJ C00193 BC00193 VJ=50.00  +MOVJ EC00193 VJ=50.00
MOVL C00194 BC00194 V=400.0  +MOVJ EC00194 VJ=100.00
MOVL C00195 BC00195 V=400.0  +MOVJ EC00195 VJ=100.00
MOVL C00196 BC00196 V=400.0  +MOVJ EC00196 VJ=100.00
MOVL C00197 BC00197 V=400.0  +MOVJ EC00197 VJ=100.00
MOVL C00198 BC00198 V=400.0  +MOVJ EC00198 VJ=100.00
MOVL C00199 BC00199 V=400.0  +MOVJ EC00199 VJ=100.00
SFTON3D P054
SMOVL C00200 BC00200 V=133.3 PL=0  +MOVJ EC00200
SREFP 1 C00201 BC00201  +REFP EC00201
SREFP 2 C00202 BC00202  +REFP EC00202
MACRO1 MJ#(0) ARGF14
ARCON
SFTON3D P055
SMOVL C00203 BC00203 V=11.7  +MOVJ EC00203
SMOVL C00204 BC00204 V=11.7  +MOVJ EC00204
SMOVL C00205 BC00205 V=11.7  +MOVJ EC00205
ARCOF
SMOVL C00206 BC00206 V=166.7  +MOVJ EC00206
SMOVL C00207 BC00207 V=400.0  +MOVJ EC00207
SFTOF3D
SMOVL C00208 BC00208 V=400.0  +MOVJ EC00208
SMOVL C00209 BC00209 V=400.0  +MOVJ EC00209
SMOVL C00210 BC00210 V=400.0  +MOVJ EC00210
SMOVL C00211 BC00211 V=400.0  +MOVJ EC00211
SFTON3D P052
SMOVL C00212 BC00212 V=133.3 PL=0  +MOVJ EC00212
SREFP 1 C00213 BC00213  +REFP EC00213
SREFP 2 C00214 BC00214  +REFP EC00214
ARCON
SFTON3D P051
SMOVL C00215 BC00215 V=11.7  +MOVJ EC00215
SMOVL C00216 BC00216 V=11.7  +MOVJ EC00216
SMOVL C00217 BC00217 V=11.7  +MOVJ EC00217
SMOVL C00218 BC00218 V=11.7  +MOVJ EC00218
ARCOF
SMOVL C00219 BC00219 V=166.7  +MOVJ EC00219
SFTOF3D
SMOVL C00220 BC00220 V=400.0  +MOVJ EC00220
SMOVL C00221 BC00221 V=400.0  +MOVJ EC00221
SMOVL C00222 BC00222 V=400.0  +MOVJ EC00222
SMOVL C00223 BC00223 V=400.0  +MOVJ EC00223
SMOVL C00224 BC00224 V=400.0  +MOVJ EC00224
SMOVL C00225 BC00225 V=400.0  +MOVJ EC00225
SMOVL C00226 BC00226 V=400.0  +MOVJ EC00226
SFTON3D P054
SMOVL C00227 BC00227 V=133.3 PL=0  +MOVJ EC00227
ARCON
SMOVL C00228 BC00228 V=11.7  +MOVJ EC00228
SFTON3D P053
SMOVL C00229 BC00229 V=11.7  +MOVJ EC00229
ARCOF
SMOVL C00230 BC00230 V=400.0  +MOVJ EC00230
SFTOF3D
SMOVL C00231 BC00231 V=400.0  +MOVJ EC00231
SMOVL C00232 BC00232 V=400.0  +MOVJ EC00232
SMOVL C00233 BC00233 V=666.7  +MOVJ EC00233
SMOVL C00234 BC00234 V=666.7  +MOVJ EC00234
SMOVL C00235 BC00235 V=400.0  +MOVJ EC00235
SFTON3D P052
SMOVL C00236 BC00236 V=133.3 PL=0  +MOVJ EC00236
ARCON
SMOVL C00237 BC00237 V=11.7  +MOVJ EC00237
SFTON3D P053
SMOVL C00238 BC00238 V=11.7  +MOVJ EC00238
SMOVL C00239 BC00239 V=11.7  +MOVJ EC00239
ARCOF
SMOVL C00240 BC00240 V=166.7  +MOVJ EC00240
SFTOF3D
SMOVL C00241 BC00241 V=400.0  +MOVJ EC00241
SMOVL C00242 BC00242 V=400.0  +MOVJ EC00242
SMOVL C00243 BC00243 V=666.7  +MOVJ EC00243
'Path W1425
SFTOF3D
SFTON3D P023
MOVJ C00244 BC00244 VJ=100.00  +MOVJ EC00244 VJ=100.00
SMOVL C00245 BC00245 V=166.7  +MOVJ EC00245
SMOVL C00246 BC00246 V=133.3 PL=0  +MOVJ EC00246
SREFP 1 C00247 BC00247  +REFP EC00247
SREFP 2 C00248 BC00248  +REFP EC00248
MACRO1 MJ#(0) ARGF14
ARCON
SMOVL C00249 BC00249 V=10.0  +MOVJ EC00249
ARCOF
SMOVL C00250 BC00250 V=400.0  +MOVJ EC00250
SMOVL C00251 BC00251 V=1000.0  +MOVJ EC00251
SFTOF3D
'Path W1426
SFTOF3D
SFTON3D P022
MOVJ C00252 BC00252 VJ=100.00  +MOVJ EC00252 VJ=100.00
SMOVL C00253 BC00253 V=133.3 PL=0  +MOVJ EC00253
SREFP 1 C00254 BC00254  +REFP EC00254
SREFP 2 C00255 BC00255  +REFP EC00255
MACRO1 MJ#(0) ARGF14
ARCON
SMOVL C00256 BC00256 V=10.0  +MOVJ EC00256
ARCOF
SMOVL C00257 BC00257 V=400.0  +MOVJ EC00257
SMOVL C00258 BC00258 V=1000.0  +MOVJ EC00258
SFTOF3D
'Path W1427
SFTOF3D
SFTON3D P021
MOVJ C00259 BC00259 VJ=100.00  +MOVJ EC00259 VJ=100.00
SMOVL C00260 BC00260 V=133.3 PL=0  +MOVJ EC00260
SREFP 1 C00261 BC00261  +REFP EC00261
SREFP 2 C00262 BC00262  +REFP EC00262
MACRO1 MJ#(0) ARGF14
ARCON
SMOVL C00263 BC00263 V=10.0  +MOVJ EC00263
ARCOF
SMOVL C00264 BC00264 V=400.0  +MOVJ EC00264
SFTOF3D
MOVJ C00265 BC00265 VJ=100.00  +MOVJ EC00265 VJ=100.00
MOVJ C00266 BC00266 VJ=100.00  +MOVJ EC00266 VJ=100.00
MOVJ C00267 BC00267 VJ=100.00  +MOVJ EC00267 VJ=100.00
END
